TYPE ST_CURING_STATION_HEATER_CONTROL_STATE :
STRUCT
	enabled:					BOOL;
	heat:						BOOL;
	fan:						BOOL;
	tempInC:					REAL;
//		tempInF:					REAL;
	testTemperatureReached:		BOOL; 
	workTemperatureReached:		BOOL;
	stationId:					UDINT; 
END_STRUCT
END_TYPE

(* stored: Version 1.1.0.1
   DUT ST_CURING_STATION_HEATER_CONTROL_STATE: Id {15b71431-4699-4e45-ae28-f1cd8c1b9efa} *)
